FUNCTION_BLOCK MessageEventLogger IMPLEMENTS Message
VAR
	message : FB_TcMessage;
	_Source : Name;
END_VAR

PROPERTY Arguments : I_TcArguments
GET
Arguments := message.ipArguments;
END_GET
END_PROPERTY

METHOD ClearArguments : I_TcArguments
message.ipArguments.Clear();

IF (_Source <> 0) THEN
	message.ipArguments.AddStringByValue(value := _Source.Name);
END_IF

ClearArguments := message.ipArguments;
END_METHOD

METHOD FB_init : BOOL
VAR_INPUT
	bInitRetains : BOOL; // if TRUE, the retain variables are initialized (warm start / cold start)
	bInCopyCode : BOOL;  // if TRUE, the instance afterwards gets moved into the copy code (online change)
	
	event : TcEventEntry;
END_VAR
message.CreateEx(stEventEntry := event, ipSourceInfo := 0);
END_METHOD

METHOD Send
VAR_INPUT
END_VAR
IF (message.ipArguments.nCount = 0 AND _Source <> 0) THEN
	message.ipArguments.AddStringByValue(value := _Source.Name);
END_IF

message.Send(0);
END_METHOD

{attribute 'monitoring' := 'call'}
PROPERTY Source : Name
GET
Source := _Source;
END_GET
SET
_Source := Source;
END_SET
END_PROPERTY

METHOD Watch
VAR_INPUT
	eventCondition : BOOL;
END_VAR
IF (eventCondition) THEN
	Send();
END_IF
END_METHOD

END_FUNCTION_BLOCK

(* stored: Version 1.1.0.1
   POU MessageEventLogger: Id {c65b3b8c-cefe-0c69-28d9-e22d6f05aacc}, SpecialFunc None
   Property Arguments: Id {a4cdc9b9-9175-0235-24d3-9175fa50c141}
   Get Get: Id {0d2cf21f-7a2a-0f95-3410-db23e36240a7}
   Method ClearArguments: Id {572aa0f7-ae4e-0bbe-06b8-619f0b33aaaf}
   Method FB_init: Id {bd18aeaa-a101-03cb-0902-b738f218667a}
   Method Send: Id {f0733f31-9e20-025f-2b59-69033ef37c10}
   Property Source: Id {85dd2fb6-f7e3-028b-0d93-8fe6326af09f}
   Get Get: Id {f3ba702f-40d7-0e55-0ef0-b6d2b973d449}
   Set Set: Id {a5a22b04-d5b2-0c00-0bc9-9a1597efe5ae}
   Method Watch: Id {56e12bb0-a397-01d5-1032-1331946bc7c3} *)
